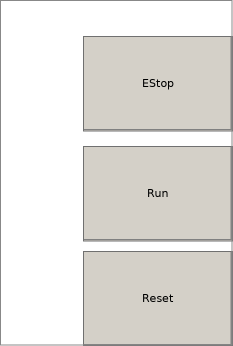
VISUALIZATION Visualization  // 233x346
    Button (83,36 150x95), "EStop"
        toggle MAIN.HMI_EStop
    Button (83,146 150x95), "Run"
        toggle MAIN.HMI_Run
    Button (83,251 150x95), "Reset"
        tap MAIN.HMI_Restart p1329445385=TRUE
END_VISUALIZATION

(* stored: Version 1.1.0.1
   Visu Visualization: Id {ea1bbd13-d2ab-4419-9642-7346f6f08260} *)
